// SIMATIC S7-200 project (STEP 7-Micro/WIN), CPU 221 REL 01.10

SYMBOL_TABLE USER1
tang1            M0.0
tang2            M0.1
tang3            M0.2
tang4            M0.4
start            I0.0
stopp            I0.1
cb1              I0.2
cb2              I0.3
van              Q0.0
dc1              Q0.1
dc2              Q0.2
dong_co_khuay    Q0.3
END_SYMBOL_TABLE

ORGANIZATION_BLOCK MAIN:OB1
TITLE=PROGRAM COMMENTS
BEGIN
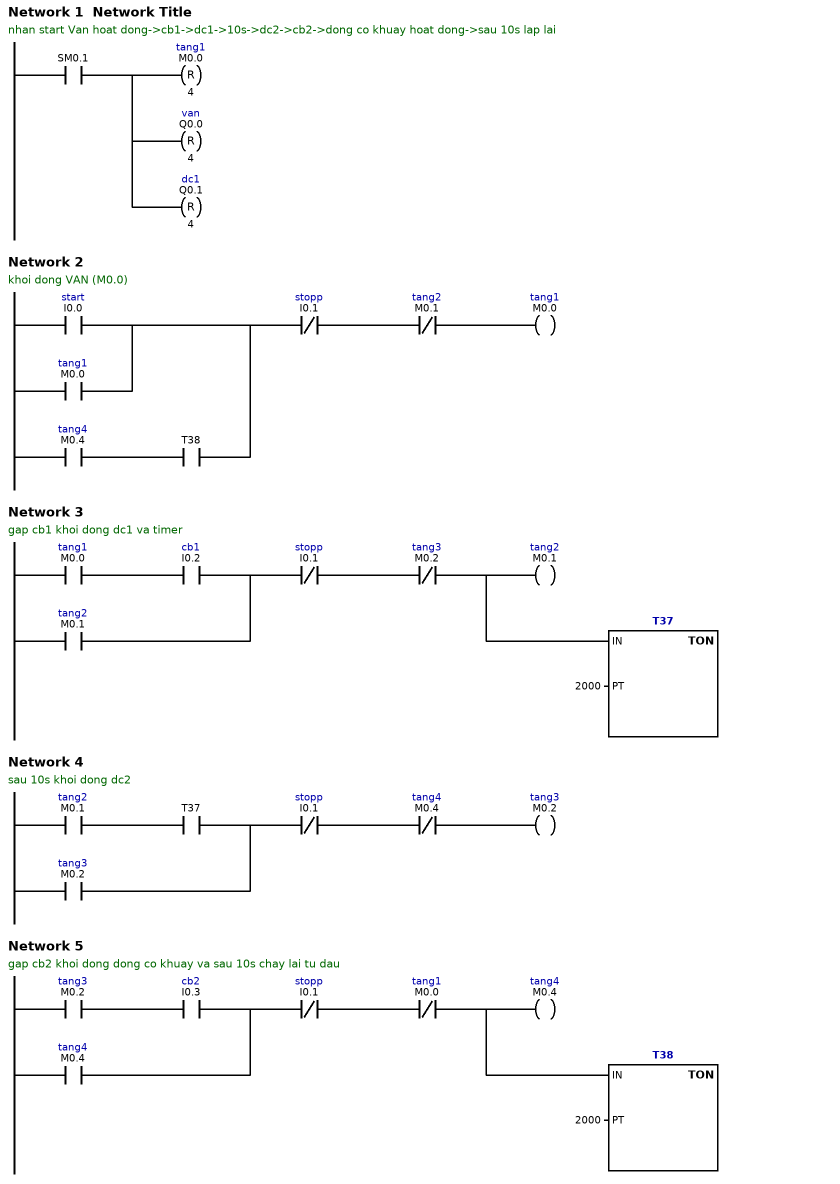
Network 1 // Network Title
// nhan start Van hoat dong->cb1->dc1->10s->dc2->cb2->dong co khuay hoat dong->sau 10s lap lai
LD     SM0.1
R      tang1:M0.0, 4
R      van:Q0.0, 4
R      dc1:Q0.1, 4
Network 2
// khoi dong VAN (M0.0)
LD     start:I0.0
O      tang1:M0.0
LD     tang4:M0.4
A      T38
OLD
AN     stopp:I0.1
AN     tang2:M0.1
=      tang1:M0.0
Network 3
// gap cb1 khoi dong dc1 va timer
LD     tang1:M0.0
A      cb1:I0.2
O      tang2:M0.1
AN     stopp:I0.1
AN     tang3:M0.2
=      tang2:M0.1
TON    T37, 2000
Network 4
// sau 10s khoi dong dc2
LD     tang2:M0.1
A      T37
O      tang3:M0.2
AN     stopp:I0.1
AN     tang4:M0.4
=      tang3:M0.2
Network 5
// gap cb2 khoi dong dong co khuay va sau 10s chay lai tu dau
LD     tang3:M0.2
A      cb2:I0.3
O      tang4:M0.4
AN     stopp:I0.1
AN     tang1:M0.0
=      tang4:M0.4
TON    T38, 2000
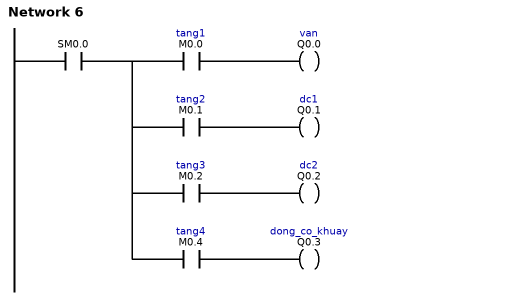
Network 6
LD     SM0.0
LPS
A      tang1:M0.0
=      van:Q0.0
LRD
A      tang2:M0.1
=      dc1:Q0.1
LRD
A      tang3:M0.2
=      dc2:Q0.2
LPP
A      tang4:M0.4
=      dong_co_khuay:Q0.3
END_ORGANIZATION_BLOCK
